{attribute 'qualified_only'}
{attribute 'strict'}
TYPE E_LAMP_STATUS :
(
	OK	:= 0,
	ERROR
);
END_TYPE

(* stored: Version 1.1.0.1, ProductVersion 3.1.4022.16
   DUT E_LAMP_STATUS: Id {9228767e-d8a5-48e9-8d13-53c033240d98} *)
